(*
SPDX-FileCopyrightText: © 2026 Oleksandr Tiutyk <trofimich@gmail.com>
SPDX-License-Identifier: MIT
License: https://opensource.org/license/mit
*)

(*!
<summary>Reports an unsupported operation using a caller-supplied message.</summary>
<description>
Diagnostic string inputs are borrowed only during the call; retained diagnostic text is copied into owned
storage. Dynamic copies are explicitly registered by Clone after construction; plain __NEW does not transfer
ownership to the task manager.
</description>
*)

{attribute 'enable_dynamic_creation'}
{attribute 'no_explicit_call' := 'do not call this function block directly'}
FUNCTION_BLOCK NotSupportedException EXTENDS GeneralException IMPLEMENTS INotSupportedException
VAR_STAT
	//! <summary>Class name shared by all instances of this function block.</summary>
	{attribute 'hide'} 
	_ClassName : STRING := __POUNAME();
END_VAR

{attribute 'monitoring' := 'call'}
PROPERTY ClassName : REFERENCE TO STRING
GET
ClassName REF= _ClassName;
END_GET
END_PROPERTY

(*!
<summary>Creates a clone of this concrete exception type.</summary>
<description>
Copies GeneralException fields and timestamps. DynamicMemoryManager owns the clone until cleanup of the
creating task; callers must not delete it. Allocation failure is terminal. Registers the newly constructed
instance before copying payload, outside FB_init. Registration failure releases the unregistered instance and
raises a terminal error; copy failure leaves the registered instance owned by the task manager for cleanup.
Custom overrides must follow the same ownership sequence.
</description>
*)
METHOD Clone : IObject
VAR
	exceptionClone : POINTER TO NotSupportedException;
END_VAR
exceptionClone := __NEW(NotSupportedException);

IF exceptionClone = 0 THEN
	DynamicMemoryManager.RaiseAllocationFailure();
END_IF

DynamicMemoryManager.RegisterAutoDisposedObject(autoDisposedObject := exceptionClone^);

exceptionClone^.CopyGeneralFields(sourceException := THIS^);

Clone := exceptionClone^;
END_METHOD

(*!
<summary>Provides the library namespace used in diagnostics.</summary>
<description>
Borrowed read-only reference to the compiler-initialized library namespace; no ownership transfer.
</description>
*)
{attribute 'monitoring' := 'call'}
PROPERTY NamespaceName : REFERENCE TO STRING
GET
NamespaceName REF= CurrentNamespace.Name;
END_GET
END_PROPERTY

(*!
<summary>Reports the byte size of this concrete instance.</summary>
<description>
Uses XSIZEOF on the instance. Does not include separately allocated payloads or prove that an arbitrary
address is valid.
</description>
*)
{attribute 'monitoring' := 'call'}
PROPERTY SelfSize : ULINT
GET
SelfSize := XSIZEOF(THIS^);
END_GET
END_PROPERTY

(*!
<summary>Raises an unsupported-operation exception with the supplied diagnostic.</summary>
<description>
Long diagnostic strings are borrowed read-only for this call; their references are not retained. Pass
variables or literals, and store computed expressions in local variables before calling. The caller must
supply a nonempty message; this precondition is not checked at runtime.
</description>
*)
METHOD Throw
VAR_INPUT
	sourceNamespaceName : STRING;
	sourceClassName : STRING;
	sourcePOUName : STRING;
	sourcePosition : STRING;
END_VAR
VAR_IN_OUT CONSTANT
	message : ERROR_MESSAGE;
END_VAR
InternalThrow(
	sourceNamespaceName := sourceNamespaceName,
	sourceClassName := sourceClassName,
	sourcePOUName := sourcePOUName,
	sourcePosition := sourcePosition,
	message := message,
	errorCode := 0,
	innerException := 0
);
END_METHOD

END_FUNCTION_BLOCK

(* stored: Version 1.1.0.1
   POU NotSupportedException: Id {ca8720a5-ceb8-45cd-a5ed-242709c5f465}, SpecialFunc None
   Property ClassName: Id {fa308b47-165a-4d2c-b0e0-96bb0f0311bf}
   Get Get: Id {2b32fbdb-997b-4572-8009-392deb237a2e}
   Method Clone: Id {b049cd35-bfc4-4bc2-b2a8-87cab0b092ff}
   Property NamespaceName: Id {88785400-5425-4442-994b-d0dee3124a0a}
   Get Get: Id {2c990c16-8087-43bf-af3b-67fd1502e142}
   Property SelfSize: Id {80ce1cde-f861-4c75-b814-e388e2b58a2f}
   Get Get: Id {f74f64e8-7d99-41a1-a696-ef463556d251}
   Method Throw: Id {4f1e3799-83c4-482e-bcef-2e46b0881cf9} *)
